FUNCTION_BLOCK IncorrectTypeDeserializationError_TestSuite EXTENDS TcUnit.FB_TestSuite

TestAccept();
TestErrorType();
TestIsSameAsWithSameErrors();
TestIsSameAsWithDifferentErrors();
TestMessage();
TestSerializeWith();

METHOD PUBLIC TestAccept
VAR
	error : IncorrectTypeDeserializationError('testType');
	visitor : MockErrorVisitor(ExpectedError := error);
END_VAR
TEST('TestAccept');

error.Accept(visitor);

AssertTrue(
	Condition := visitor.VisitedCorrectError,
	Message := 'Did not invoke VisitError on the visitor'
);

TEST_FINISHED();
END_METHOD

METHOD PUBLIC TestErrorType
VAR
	error : IncorrectTypeDeserializationError('testType');
END_VAR
TEST('TestErrorType');

AssertEquals_String(
	Actual := error.ErrorType,
	Expected := 'INCORRECT_DATATYPE_DESERIALIZATION_ERROR',
	Message := 'Did not return the expected ErrorType'
);

TEST_FINISHED();
END_METHOD

METHOD PUBLIC TestIsSameAsWithDifferentErrors
VAR
	error1 : IncorrectTypeDeserializationError('testType');
	error2 : MockError(MockErrorType:='ERROR_TYPE_B',MockMessage:='Message 2');
END_VAR
TEST('TestIsSameAsWithDifferentErrors');

AssertFalse(
	Condition := error1.IsSameAs(error2),
	Message := 'Did not correctly identify errors as being different type'
);

TEST_FINISHED();
END_METHOD

METHOD PUBLIC TestIsSameAsWithSameErrors
VAR
	error1 : IncorrectTypeDeserializationError('testType');
	error2 : MockError(MockErrorType:='INCORRECT_DATATYPE_DESERIALIZATION_ERROR',MockMessage:='Message');
END_VAR
TEST('TestIsSameAsWithSameErrors');

AssertTrue(
	Condition := error1.IsSameAs(error2),
	Message := 'Did not correctly identify errors as being the same type'
);

TEST_FINISHED();
END_METHOD

METHOD PUBLIC TestMessage
VAR
	error : IncorrectTypeDeserializationError('testType');
END_VAR
TEST('TestMessage');

AssertEquals_String(
	Actual := error.Message,
	Expected := 'Deserialization Failed, Incorrect Datatype : testType',
	Message := 'Did not return the expected Message'
);

TEST_FINISHED();
END_METHOD

METHOD PUBLIC TestSerializeWith
VAR
	error : IncorrectTypeDeserializationError('testType');
	serializer : MockJsonSerializer;
	result : T_MAXSTRING;
END_VAR
TEST('TestSerializeWith');

error.SerializeWith(serializer);
serializer.TryGetSerializedData(ADR(result), SIZEOF(result));

AssertEquals_String(
	Actual := result,
	Expected := '{"errorType":"INCORRECT_DATATYPE_DESERIALIZATION_ERROR","message":"Deserialization Failed, Incorrect Datatype : testType"}',
	Message := 'Did not serialize correctly'
);

TEST_FINISHED();
END_METHOD

END_FUNCTION_BLOCK

(* stored: Version 1.1.0.1, ProductVersion 3.1.4024.12
   POU IncorrectTypeDeserializationError_TestSuite: Id {84c55437-edee-4a79-babb-3090c3890166}, SpecialFunc None
   Method TestAccept: Id {1ea8d6e3-b81c-4b50-b2a7-1b196a76bd5c}
   Method TestErrorType: Id {a2b171b7-3bac-454b-9dc4-035376d381c7}
   Method TestIsSameAsWithDifferentErrors: Id {23c49470-5c9c-400e-b672-5c612a1887c6}
   Method TestIsSameAsWithSameErrors: Id {cf58a995-db94-4a10-8fe7-12f28867d80a}
   Method TestMessage: Id {e2cdfef9-eef9-45f9-a025-12f99889bf9b}
   Method TestSerializeWith: Id {fe9025a8-6e32-4f9a-ba1a-c736da496af9} *)
